(* IEC 61131-3 sources: eebus-docker-bridge/Codesys, 3 files *)

(* ---- eLpcZustand.st ---- *)
// Zustand des Use Case LPC, wie ihn die EEBUS-Brücke meldet.
// Zahlenwerte identisch mit LpcZustand in bruecke.go.
{attribute 'qualified_only'}
{attribute 'strict'}
TYPE eLpcZustand :
(
	Init                := 0,   // nach Neustart, Failsafe-Grenze gilt
	UnbegrenztGesteuert := 1,   // Steuerbox verbunden, keine aktive Grenze
	Begrenzt            := 2,   // Grenze des Netzbetreibers aktiv
	Failsafe            := 3,   // Heartbeat ausgefallen, Failsafe-Grenze gilt
	UnbegrenztAutonom   := 4,   // keine Kommunikation, Failsafe-Mindestdauer abgelaufen
	Unbekannt           := 99   // Brücke nicht erreichbar oder Wert ungültig
) UINT;
END_TYPE

(* ---- GvlEebus.st ---- *)
// Prozessabbild der Modbus-Verbindung zur EEBUS-Brücke.
// Mapping im Gerätebaum (Modbus TCP Client -> Server 127.0.0.1:5502):
//   Kanal 1: FC04 Read Input Registers,  Offset 0, Länge 14, Zyklus 200 ms -> aInputRegister
//   Kanal 2: FC16 Write Multiple Registers, Offset 0, Länge 3,  Zyklus 1 s  -> aHoldingRegister
{attribute 'qualified_only'}
VAR_GLOBAL
	aInputRegister   : ARRAY [0..13] OF WORD;   // Brücke -> SPS
	aHoldingRegister : ARRAY [0..2] OF WORD;    // SPS -> Brücke
END_VAR

(* ---- PrgEnergiemanagement.st ---- *)
// Beispielaufruf. Die Aufteilung der Grenze auf die einzelnen steuerbaren
// Verbraucher (Wallboxen, Wärmepumpe, ...) ist anlagenspezifisch.
PROGRAM PrgEnergiemanagement
VAR
	fbEebusLpc               : FbEebusLpc;
	udiAnforderungW          : UDINT;   // ungeregelte Summenanforderung der steuerbaren Verbraucher
	udiFreigegebeneLeistungW : UDINT;   // Vorgabe an die Verteillogik
END_VAR

fbEebusLpc(
	xFreigabe           := TRUE,
	aInputRegister      := GvlEebus.aInputRegister,
	udiNennleistungMaxW := 22000,
	udiErsatzgrenzeW    := 4200,
	tBrueckeTimeout     := T#10S);

GvlEebus.aHoldingRegister := fbEebusLpc.aHoldingRegister;

IF fbEebusLpc.xBegrenzungAktiv THEN
	udiFreigegebeneLeistungW := MIN(udiAnforderungW, fbEebusLpc.udiLeistungsgrenzeW);
ELSE
	udiFreigegebeneLeistungW := udiAnforderungW;
END_IF
END_PROGRAM
